% RSLogix 500 project P8_IVANOVSKI_M.RSS, saved by version 8.30.00.16 %
PROJECT "UNTITLED"    % processor: Bul.1763 MicroLogix 1100 Series B %

PROGRAM FILES
  LAD 2 "MAIN"  3 rungs
  LAD 3 "IO/MEMORY"  2 rungs
  LAD 4 "CONTROLS"  4 rungs

DATA FILES
  O0 OUTPUT  6 elements
  I1 INPUT  12 elements
  S2 STATUS  66 elements
  B3 BINARY  2 elements
  T4 TIMER  1 elements
  C5 COUNTER  1 elements
  R6 CONTROL  1 elements
  N7 INTEGER  4 elements
  F8 FLOAT  1 elements

LADDER 2 "MAIN"
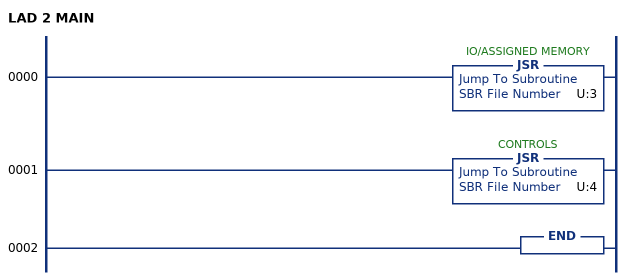
% Rung: 0 %
SOR JSR U:3 EOR
%   U:3  "IO/ASSIGNED MEMORY" %
% Rung: 1 %
SOR JSR U:4 EOR
%   U:4  "CONTROLS" %
% Rung: 2 %
SOR END EOR

LADDER 3 "IO/MEMORY"
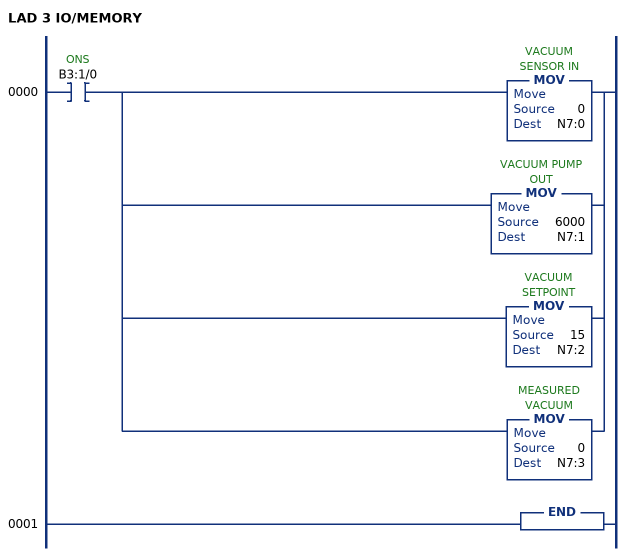
% Rung: 0 %
SOR XIC B3:1/0 BST MOV 0 N7:0 NXB MOV 6000 N7:1 NXB MOV 15 N7:2 NXB MOV 0 N7:3 BND EOR
%   B3:1/0  "ONS" %
%   N7:0  "VACUUM SENSOR IN" %
%   N7:1  "VACUUM PUMP OUT" %
%   N7:2  "VACUUM SETPOINT" %
%   N7:3  "MEASURED VACUUM" %
% Rung: 1 %
SOR END EOR

LADDER 4 "CONTROLS"
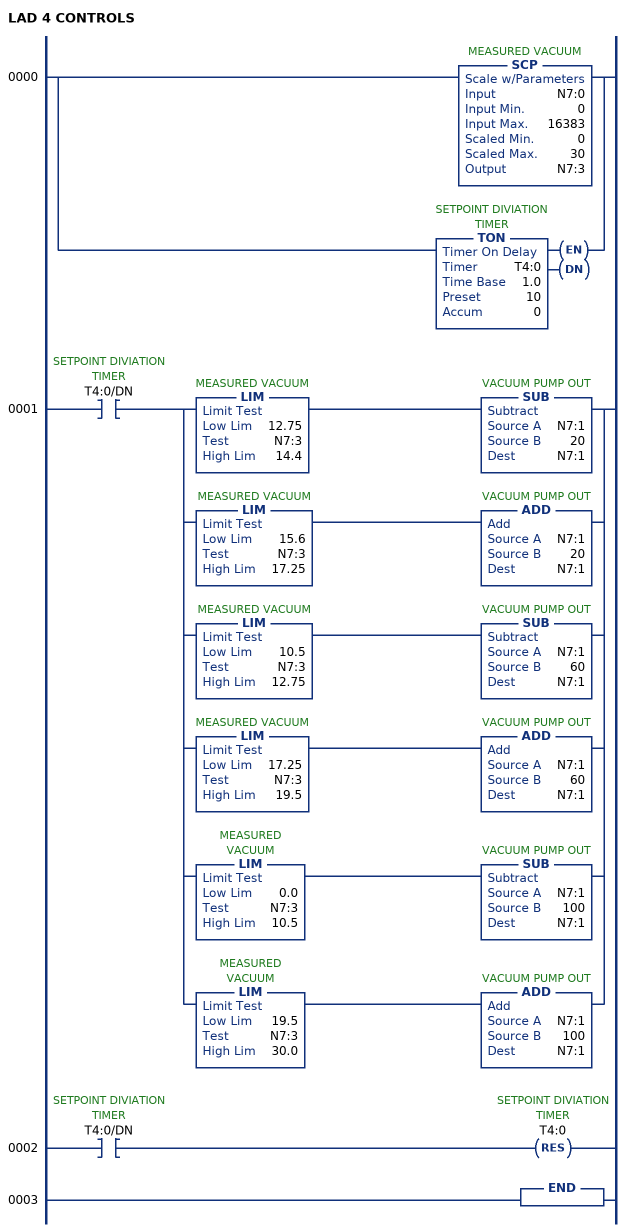
% Rung: 0 %
SOR BST SCP N7:0 0 16383 0 30 N7:3 NXB TON T4:0 1.0 10 0 BND EOR
%   N7:0  "VACUUM SENSOR IN" %
%   N7:3  "MEASURED VACUUM" %
%   T4:0  "SETPOINT DIVIATION TIMER" %
% Rung: 1 %
SOR XIC T4:0/DN BST LIM 12.75 N7:3 14.4 SUB N7:1 20 N7:1 NXB LIM 15.6 N7:3 17.25 ADD N7:1 20 N7:1 NXB LIM 10.5 N7:3 12.75 SUB N7:1 60 N7:1 NXB LIM 17.25 N7:3 19.5 ADD N7:1 60 N7:1 NXB LIM 0.0 N7:3 10.5 SUB N7:1 100 N7:1 NXB LIM 19.5 N7:3 30.0 ADD N7:1 100 N7:1 BND EOR
%   T4:0  "SETPOINT DIVIATION TIMER" %
%   N7:3  "MEASURED VACUUM" %
%   N7:1  "VACUUM PUMP OUT" %
% Rung: 2 %
SOR XIC T4:0/DN RES T4:0 EOR
%   T4:0  "SETPOINT DIVIATION TIMER" %
% Rung: 3 %
SOR END EOR

OTHER DOCUMENTED ADDRESSES
  B3:0/0  "TC #1"
  B3:0/1  "TC #2"
  B3:1/1  "ONS"
  B3:1/2  "ONS"
  B3:1/3  "ONS"
  B3:1/4  "ONS"
  B3:1/5  "ONS"
  N7:4  "VACUUM PUMP OUT"

DATA TABLE (non-zero values as saved)
DATA T4
% .PRE .ACC %
% T4:0 % 10 0
DATA N7
% N7:0 % 0 0 15 0
